FUNCTION_BLOCK Test_TimeAsString_24HourFormat EXTENDS TUnitTestBase
VAR
END_VAR

METHOD  Execute
VAR_INST
    TimeStruct : TIMESTRUCT := (wHour := 22, wMinute := 20, wSecond := 18);
END_VAR
Assertion.AssertEquals_STRING(
    Expected := '22:20:18',
    Actual   := F_TimeAsString(TimeStruct),
    ObjectName := _TestName,
    VariableName  := 'F_TimeAsString(TimeStruct)');


Test_Finished();
END_METHOD

END_FUNCTION_BLOCK

(* stored: Version 1.1.0.1, ProductVersion 3.1.4024.3
   POU Test_TimeAsString_24HourFormat: Id {22f25ef6-a0a3-4183-a54a-0750521d3582}, SpecialFunc None
   Method Execute: Id {300afb64-7e78-4bf8-aa4a-0b7c5761188c} *)
